(* Logix 5000 project; controller cal1632 1756-L62 rev 16.20; software revision 16.05; part 56 of 57 *)
(* tags used below, declared in another part *)
   FAULT : BOOL;
   HMI : BOOL;
   p01r09_pb_global_reset : BOOL;
   p30_di_pin_1 : BOOL;
   p30_di_pin_2 : BOOL;
   p30_di_pin_3 : BOOL;
   p30_di_pin_4 : BOOL;
   p30_di_pin_5 : BOOL;
   p30_di_pin_6 : BOOL;
   p30_di_pin_7 : BOOL;
   p30_di_pin_8 : BOOL;
   p30_dint_to_hmi : DINT[16];
   p30_do_retract_motion : BOOL;
   p30_do_rotation_fwd : BOOL;
   p30_do_rotation_rev : BOOL;
   p30_real_to_hmi : REAL[112];
   p30r04 : routine;
   p30r04_timer_fault : TIMER[4];
   p30r04_timer_warning : TIMER[4];
   p30r05 : routine;
   p30r05_timer_fault : TIMER[4];
   p30r05_timer_warning : TIMER[4];
   p30r06 : routine;
   p30r06_timer_fault : TIMER[4];
   p30r06_timer_warning : TIMER[4];
   p30r07 : routine;
   p30r07_timer_fault : TIMER[4];
   p30r07_timer_warning : TIMER[4];
   p30r10 : routine;
(* P30_Retraction_System, continued *)

ROUTINE R04_Output   (* ladder *)
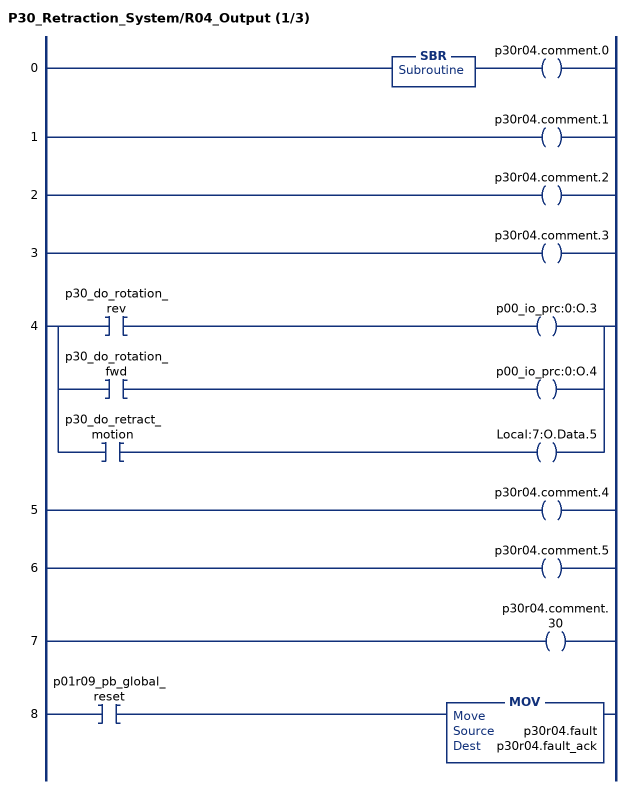
   0: SBR()OTE(p30r04.comment.0);
   1: OTE(p30r04.comment.1);
   2: OTE(p30r04.comment.2);
   3: OTE(p30r04.comment.3);
   4: [XIC(p30_do_rotation_rev) OTE(p00_io_prc:0:O.3) ,XIC(p30_do_rotation_fwd) OTE(p00_io_prc:0:O.4) ,XIC(p30_do_retract_motion) OTE(Local:7:O.Data.5) ];
   5: OTE(p30r04.comment.4);
   6: OTE(p30r04.comment.5);
   7: OTE(p30r04.comment.30);
   8: XIC(p01r09_pb_global_reset)MOV(p30r04.fault,p30r04.fault_ack);
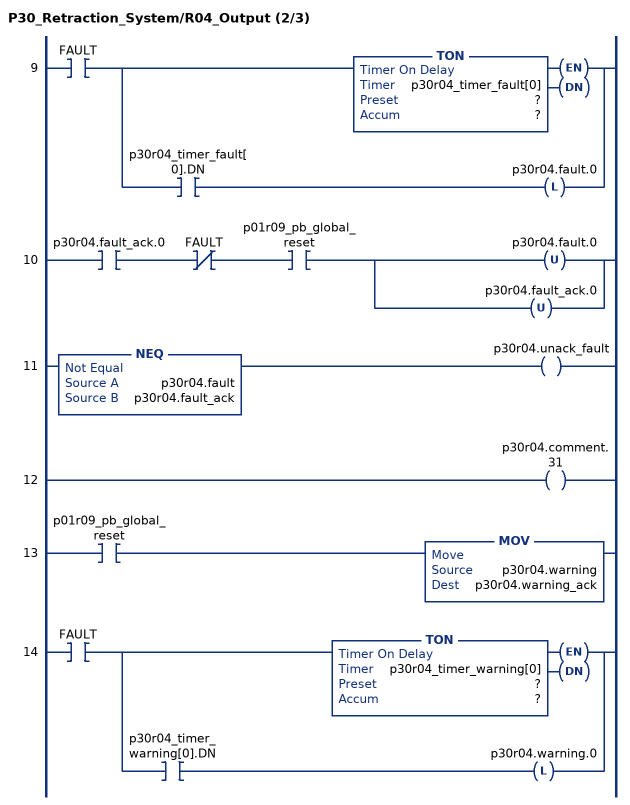
   9: XIC(FAULT)[TON(p30r04_timer_fault[0],?,?) ,XIC(p30r04_timer_fault[0].DN) OTL(p30r04.fault.0) ];
   10: XIC(p30r04.fault_ack.0)XIO(FAULT)XIC(p01r09_pb_global_reset)[OTU(p30r04.fault.0) ,OTU(p30r04.fault_ack.0) ];
   11: NEQ(p30r04.fault,p30r04.fault_ack)OTE(p30r04.unack_fault);
   12: OTE(p30r04.comment.31);
   13: XIC(p01r09_pb_global_reset)MOV(p30r04.warning,p30r04.warning_ack);
   14: XIC(FAULT)[TON(p30r04_timer_warning[0],?,?) ,XIC(p30r04_timer_warning[0].DN) OTL(p30r04.warning.0) ];
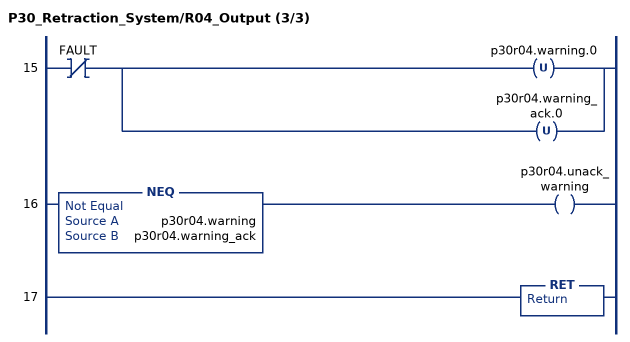
   15: XIO(FAULT)[OTU(p30r04.warning.0) ,OTU(p30r04.warning_ack.0) ];
   16: NEQ(p30r04.warning,p30r04.warning_ack)OTE(p30r04.unack_warning);
   17: RET();
END_ROUTINE

ROUTINE R05_Dint_to_HMI   (* ladder *)
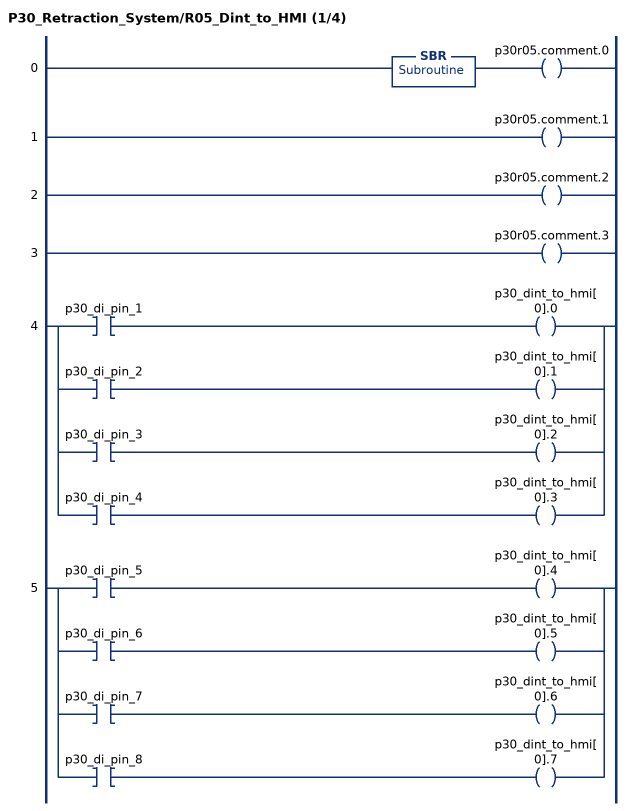
   0: SBR()OTE(p30r05.comment.0);
   1: OTE(p30r05.comment.1);
   2: OTE(p30r05.comment.2);
   3: OTE(p30r05.comment.3);
   4: [XIC(p30_di_pin_1) OTE(p30_dint_to_hmi[0].0) ,XIC(p30_di_pin_2) OTE(p30_dint_to_hmi[0].1) ,XIC(p30_di_pin_3) OTE(p30_dint_to_hmi[0].2) ,XIC(p30_di_pin_4) OTE(p30_dint_to_hmi[0].3) ];
   5: [XIC(p30_di_pin_5) OTE(p30_dint_to_hmi[0].4) ,XIC(p30_di_pin_6) OTE(p30_dint_to_hmi[0].5) ,XIC(p30_di_pin_7) OTE(p30_dint_to_hmi[0].6) ,XIC(p30_di_pin_8) OTE(p30_dint_to_hmi[0].7) ];
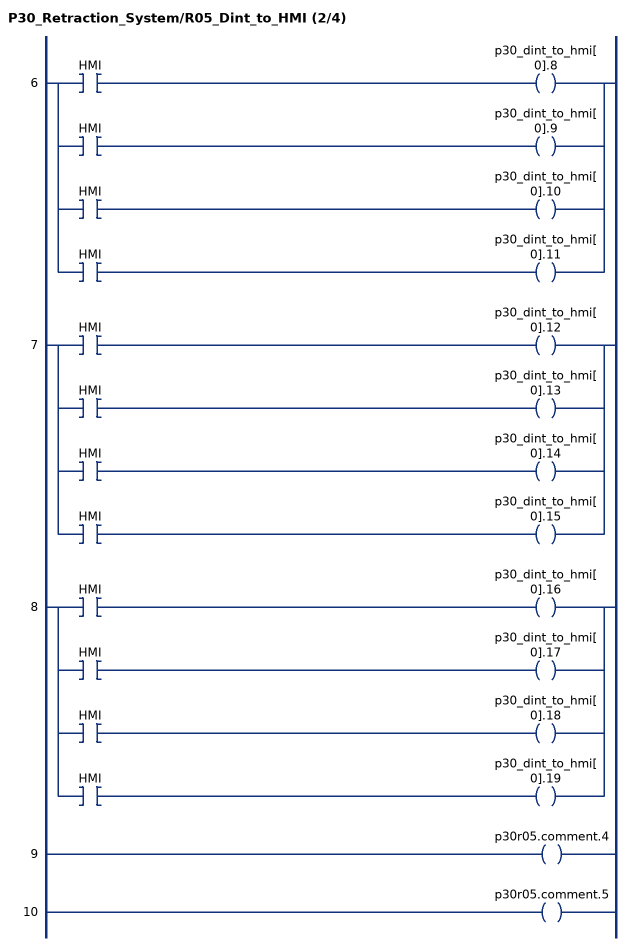
   6: [XIC(HMI) OTE(p30_dint_to_hmi[0].8) ,XIC(HMI) OTE(p30_dint_to_hmi[0].9) ,XIC(HMI) OTE(p30_dint_to_hmi[0].10) ,XIC(HMI) OTE(p30_dint_to_hmi[0].11) ];
   7: [XIC(HMI) OTE(p30_dint_to_hmi[0].12) ,XIC(HMI) OTE(p30_dint_to_hmi[0].13) ,XIC(HMI) OTE(p30_dint_to_hmi[0].14) ,XIC(HMI) OTE(p30_dint_to_hmi[0].15) ];
   8: [XIC(HMI) OTE(p30_dint_to_hmi[0].16) ,XIC(HMI) OTE(p30_dint_to_hmi[0].17) ,XIC(HMI) OTE(p30_dint_to_hmi[0].18) ,XIC(HMI) OTE(p30_dint_to_hmi[0].19) ];
   9: OTE(p30r05.comment.4);
   10: OTE(p30r05.comment.5);
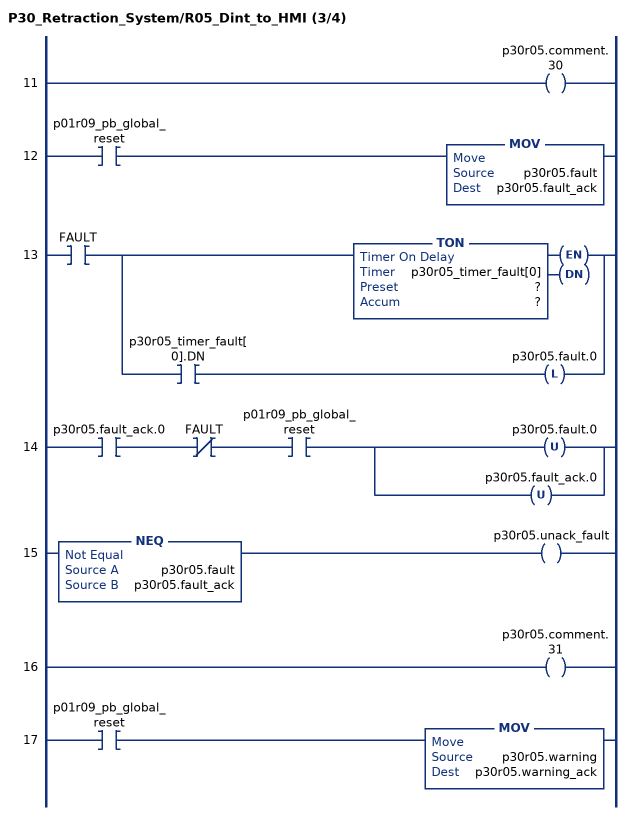
   11: OTE(p30r05.comment.30);
   12: XIC(p01r09_pb_global_reset)MOV(p30r05.fault,p30r05.fault_ack);
   13: XIC(FAULT)[TON(p30r05_timer_fault[0],?,?) ,XIC(p30r05_timer_fault[0].DN) OTL(p30r05.fault.0) ];
   14: XIC(p30r05.fault_ack.0)XIO(FAULT)XIC(p01r09_pb_global_reset)[OTU(p30r05.fault.0) ,OTU(p30r05.fault_ack.0) ];
   15: NEQ(p30r05.fault,p30r05.fault_ack)OTE(p30r05.unack_fault);
   16: OTE(p30r05.comment.31);
   17: XIC(p01r09_pb_global_reset)MOV(p30r05.warning,p30r05.warning_ack);
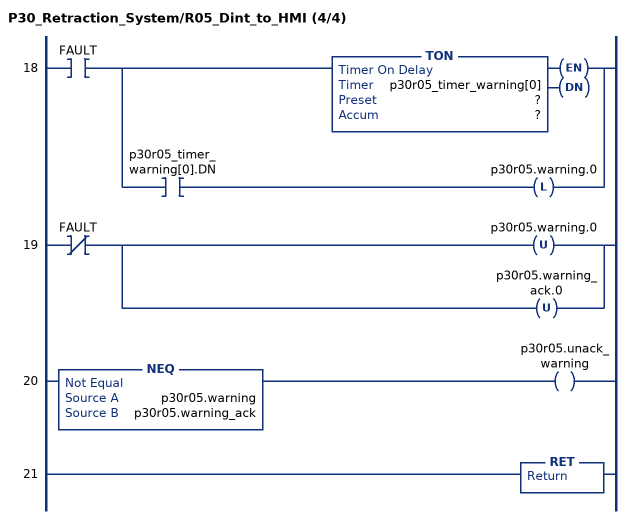
   18: XIC(FAULT)[TON(p30r05_timer_warning[0],?,?) ,XIC(p30r05_timer_warning[0].DN) OTL(p30r05.warning.0) ];
   19: XIO(FAULT)[OTU(p30r05.warning.0) ,OTU(p30r05.warning_ack.0) ];
   20: NEQ(p30r05.warning,p30r05.warning_ack)OTE(p30r05.unack_warning);
   21: RET();
END_ROUTINE

ROUTINE R06_Real_to_HMI   (* ladder *)
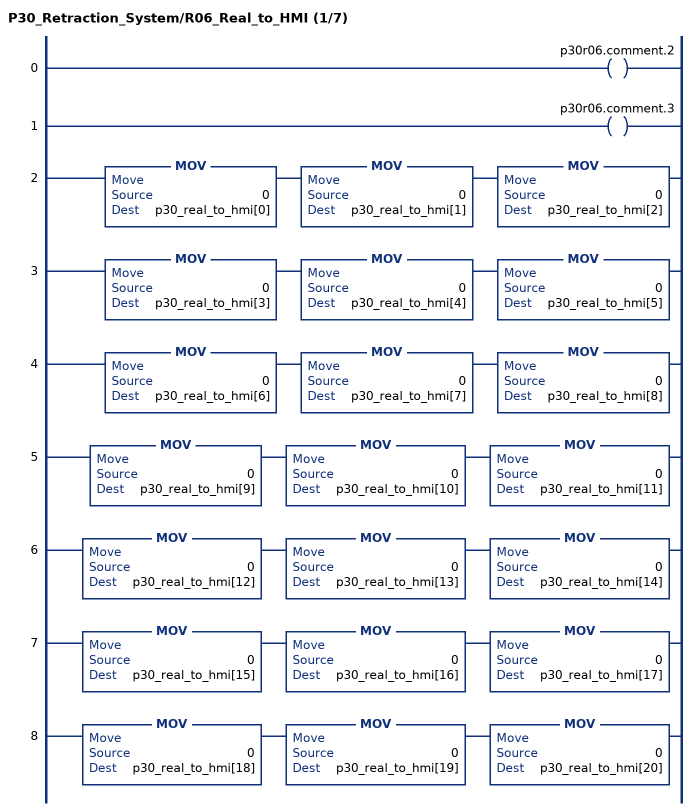
   0: OTE(p30r06.comment.2);
   1: OTE(p30r06.comment.3);
   2: MOV(0,p30_real_to_hmi[0])MOV(0,p30_real_to_hmi[1])MOV(0,p30_real_to_hmi[2]);
   3: MOV(0,p30_real_to_hmi[3])MOV(0,p30_real_to_hmi[4])MOV(0,p30_real_to_hmi[5]);
   4: MOV(0,p30_real_to_hmi[6])MOV(0,p30_real_to_hmi[7])MOV(0,p30_real_to_hmi[8]);
   5: MOV(0,p30_real_to_hmi[9])MOV(0,p30_real_to_hmi[10])MOV(0,p30_real_to_hmi[11]);
   6: MOV(0,p30_real_to_hmi[12])MOV(0,p30_real_to_hmi[13])MOV(0,p30_real_to_hmi[14]);
   7: MOV(0,p30_real_to_hmi[15])MOV(0,p30_real_to_hmi[16])MOV(0,p30_real_to_hmi[17]);
   8: MOV(0,p30_real_to_hmi[18])MOV(0,p30_real_to_hmi[19])MOV(0,p30_real_to_hmi[20]);
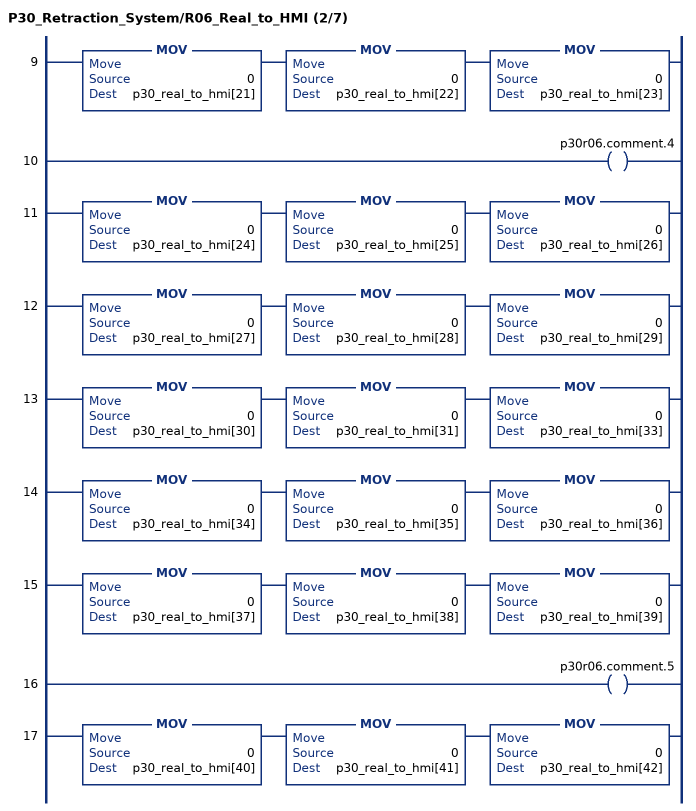
   9: MOV(0,p30_real_to_hmi[21])MOV(0,p30_real_to_hmi[22])MOV(0,p30_real_to_hmi[23]);
   10: OTE(p30r06.comment.4);
   11: MOV(0,p30_real_to_hmi[24])MOV(0,p30_real_to_hmi[25])MOV(0,p30_real_to_hmi[26]);
   12: MOV(0,p30_real_to_hmi[27])MOV(0,p30_real_to_hmi[28])MOV(0,p30_real_to_hmi[29]);
   13: MOV(0,p30_real_to_hmi[30])MOV(0,p30_real_to_hmi[31])MOV(0,p30_real_to_hmi[33]);
   14: MOV(0,p30_real_to_hmi[34])MOV(0,p30_real_to_hmi[35])MOV(0,p30_real_to_hmi[36]);
   15: MOV(0,p30_real_to_hmi[37])MOV(0,p30_real_to_hmi[38])MOV(0,p30_real_to_hmi[39]);
   16: OTE(p30r06.comment.5);
   17: MOV(0,p30_real_to_hmi[40])MOV(0,p30_real_to_hmi[41])MOV(0,p30_real_to_hmi[42]);
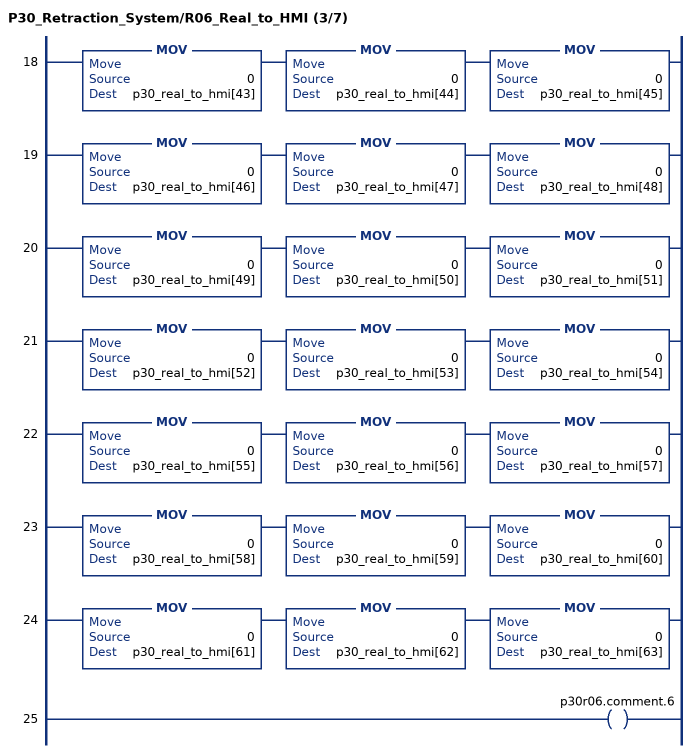
   18: MOV(0,p30_real_to_hmi[43])MOV(0,p30_real_to_hmi[44])MOV(0,p30_real_to_hmi[45]);
   19: MOV(0,p30_real_to_hmi[46])MOV(0,p30_real_to_hmi[47])MOV(0,p30_real_to_hmi[48]);
   20: MOV(0,p30_real_to_hmi[49])MOV(0,p30_real_to_hmi[50])MOV(0,p30_real_to_hmi[51]);
   21: MOV(0,p30_real_to_hmi[52])MOV(0,p30_real_to_hmi[53])MOV(0,p30_real_to_hmi[54]);
   22: MOV(0,p30_real_to_hmi[55])MOV(0,p30_real_to_hmi[56])MOV(0,p30_real_to_hmi[57]);
   23: MOV(0,p30_real_to_hmi[58])MOV(0,p30_real_to_hmi[59])MOV(0,p30_real_to_hmi[60]);
   24: MOV(0,p30_real_to_hmi[61])MOV(0,p30_real_to_hmi[62])MOV(0,p30_real_to_hmi[63]);
   25: OTE(p30r06.comment.6);
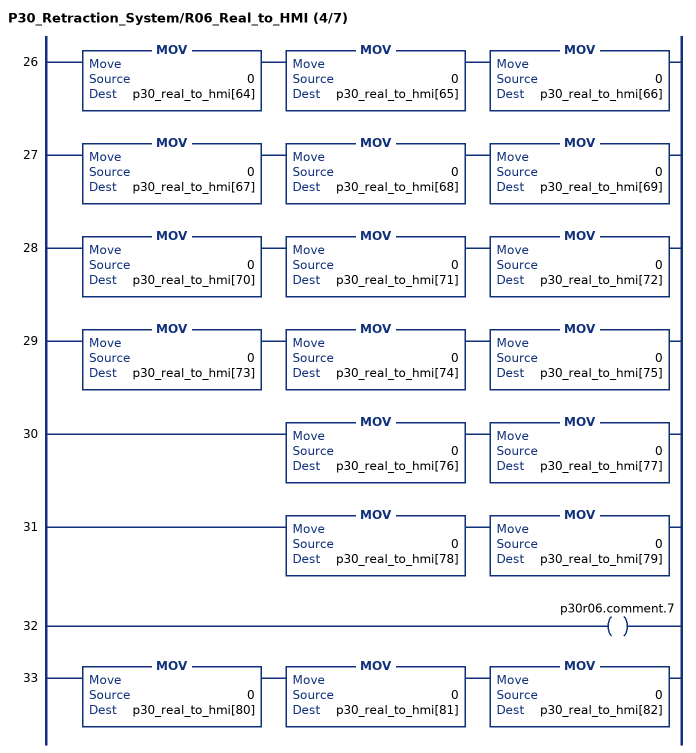
   26: MOV(0,p30_real_to_hmi[64])MOV(0,p30_real_to_hmi[65])MOV(0,p30_real_to_hmi[66]);
   27: MOV(0,p30_real_to_hmi[67])MOV(0,p30_real_to_hmi[68])MOV(0,p30_real_to_hmi[69]);
   28: MOV(0,p30_real_to_hmi[70])MOV(0,p30_real_to_hmi[71])MOV(0,p30_real_to_hmi[72]);
   29: MOV(0,p30_real_to_hmi[73])MOV(0,p30_real_to_hmi[74])MOV(0,p30_real_to_hmi[75]);
   30: MOV(0,p30_real_to_hmi[76])MOV(0,p30_real_to_hmi[77]);
   31: MOV(0,p30_real_to_hmi[78])MOV(0,p30_real_to_hmi[79]);
   32: OTE(p30r06.comment.7);
   33: MOV(0,p30_real_to_hmi[80])MOV(0,p30_real_to_hmi[81])MOV(0,p30_real_to_hmi[82]);
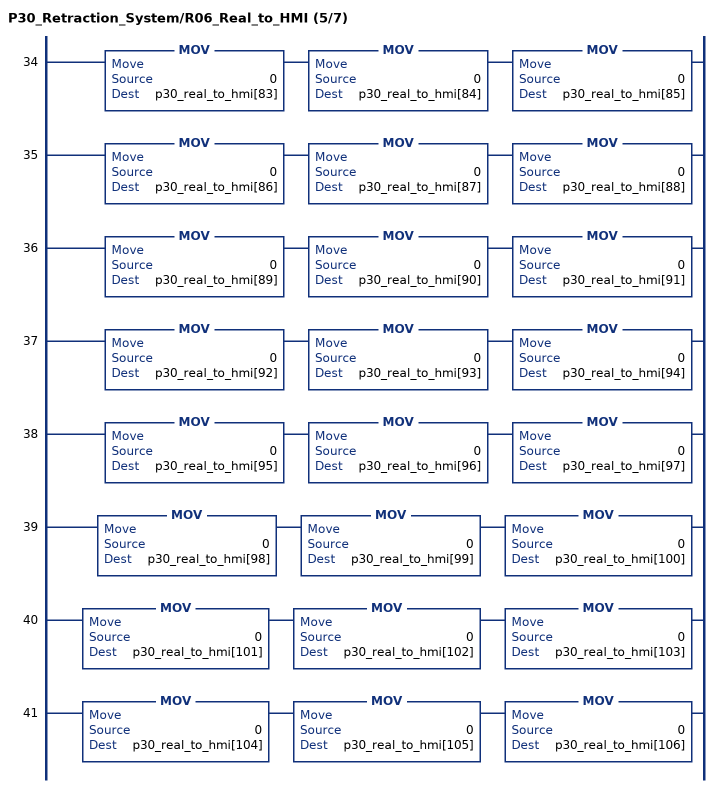
   34: MOV(0,p30_real_to_hmi[83])MOV(0,p30_real_to_hmi[84])MOV(0,p30_real_to_hmi[85]);
   35: MOV(0,p30_real_to_hmi[86])MOV(0,p30_real_to_hmi[87])MOV(0,p30_real_to_hmi[88]);
   36: MOV(0,p30_real_to_hmi[89])MOV(0,p30_real_to_hmi[90])MOV(0,p30_real_to_hmi[91]);
   37: MOV(0,p30_real_to_hmi[92])MOV(0,p30_real_to_hmi[93])MOV(0,p30_real_to_hmi[94]);
   38: MOV(0,p30_real_to_hmi[95])MOV(0,p30_real_to_hmi[96])MOV(0,p30_real_to_hmi[97]);
   39: MOV(0,p30_real_to_hmi[98])MOV(0,p30_real_to_hmi[99])MOV(0,p30_real_to_hmi[100]);
   40: MOV(0,p30_real_to_hmi[101])MOV(0,p30_real_to_hmi[102])MOV(0,p30_real_to_hmi[103]);
   41: MOV(0,p30_real_to_hmi[104])MOV(0,p30_real_to_hmi[105])MOV(0,p30_real_to_hmi[106]);
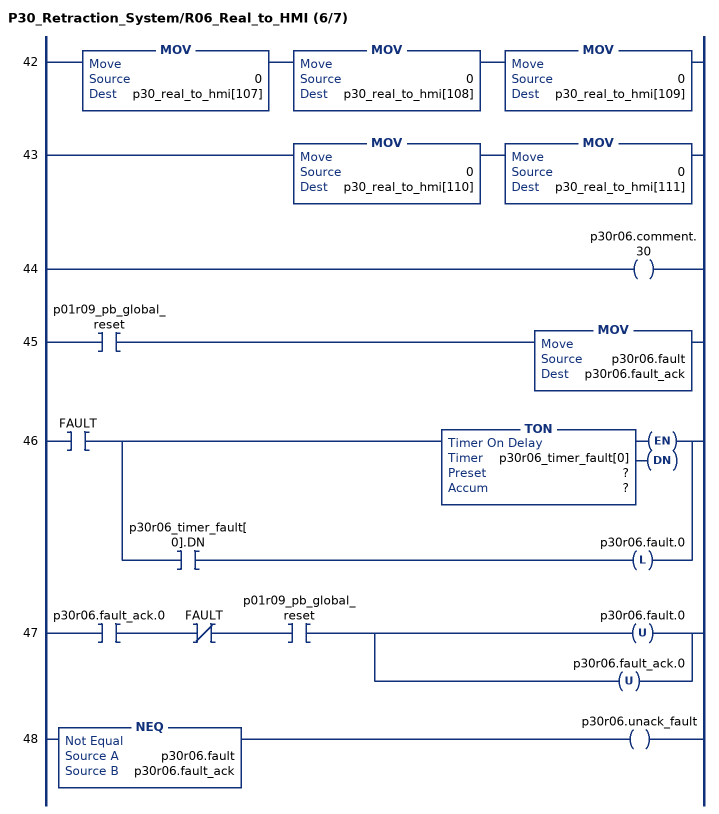
   42: MOV(0,p30_real_to_hmi[107])MOV(0,p30_real_to_hmi[108])MOV(0,p30_real_to_hmi[109]);
   43: MOV(0,p30_real_to_hmi[110])MOV(0,p30_real_to_hmi[111]);
   44: OTE(p30r06.comment.30);
   45: XIC(p01r09_pb_global_reset)MOV(p30r06.fault,p30r06.fault_ack);
   46: XIC(FAULT)[TON(p30r06_timer_fault[0],?,?) ,XIC(p30r06_timer_fault[0].DN) OTL(p30r06.fault.0) ];
   47: XIC(p30r06.fault_ack.0)XIO(FAULT)XIC(p01r09_pb_global_reset)[OTU(p30r06.fault.0) ,OTU(p30r06.fault_ack.0) ];
   48: NEQ(p30r06.fault,p30r06.fault_ack)OTE(p30r06.unack_fault);
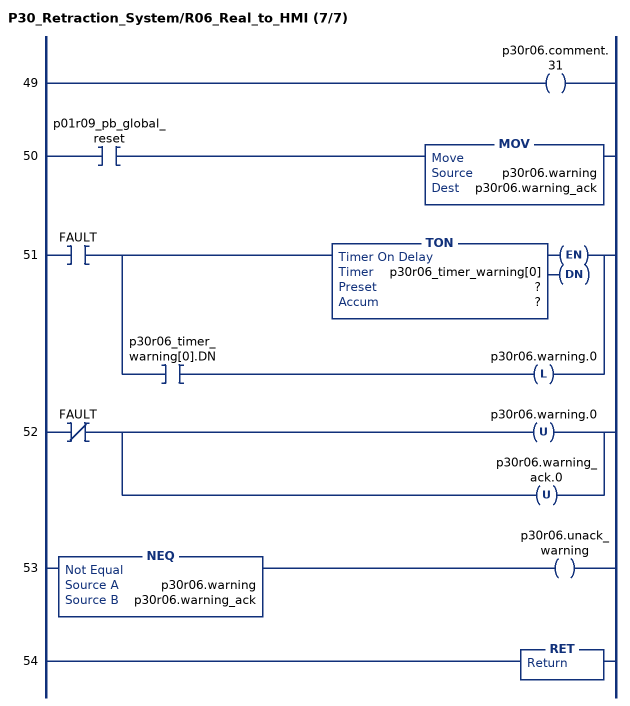
   49: OTE(p30r06.comment.31);
   50: XIC(p01r09_pb_global_reset)MOV(p30r06.warning,p30r06.warning_ack);
   51: XIC(FAULT)[TON(p30r06_timer_warning[0],?,?) ,XIC(p30r06_timer_warning[0].DN) OTL(p30r06.warning.0) ];
   52: XIO(FAULT)[OTU(p30r06.warning.0) ,OTU(p30r06.warning_ack.0) ];
   53: NEQ(p30r06.warning,p30r06.warning_ack)OTE(p30r06.unack_warning);
   54: RET();
END_ROUTINE

ROUTINE R07_Alarms   (* ladder *)
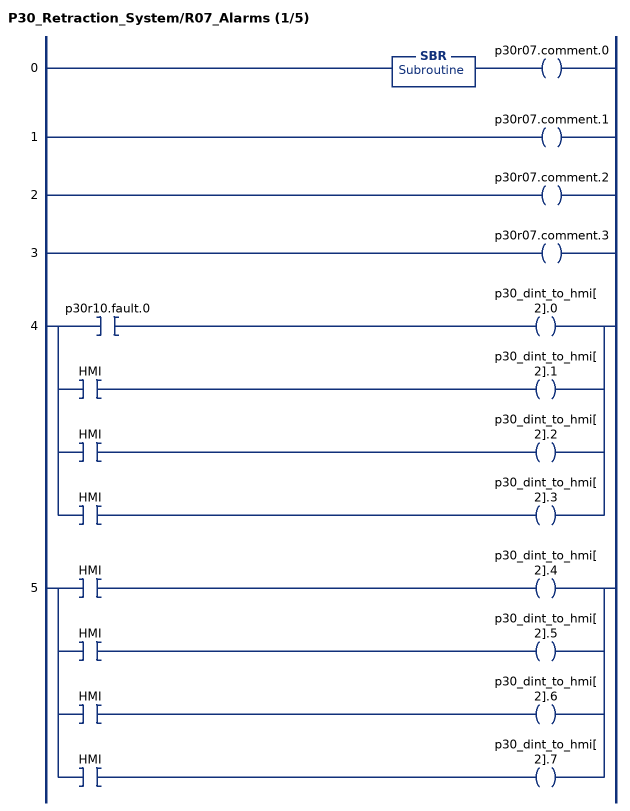
   0: SBR()OTE(p30r07.comment.0);
   1: OTE(p30r07.comment.1);
   2: OTE(p30r07.comment.2);
   3: OTE(p30r07.comment.3);
   4: [XIC(p30r10.fault.0) OTE(p30_dint_to_hmi[2].0) ,XIC(HMI) OTE(p30_dint_to_hmi[2].1) ,XIC(HMI) OTE(p30_dint_to_hmi[2].2) ,XIC(HMI) OTE(p30_dint_to_hmi[2].3) ];
   5: [XIC(HMI) OTE(p30_dint_to_hmi[2].4) ,XIC(HMI) OTE(p30_dint_to_hmi[2].5) ,XIC(HMI) OTE(p30_dint_to_hmi[2].6) ,XIC(HMI) OTE(p30_dint_to_hmi[2].7) ];
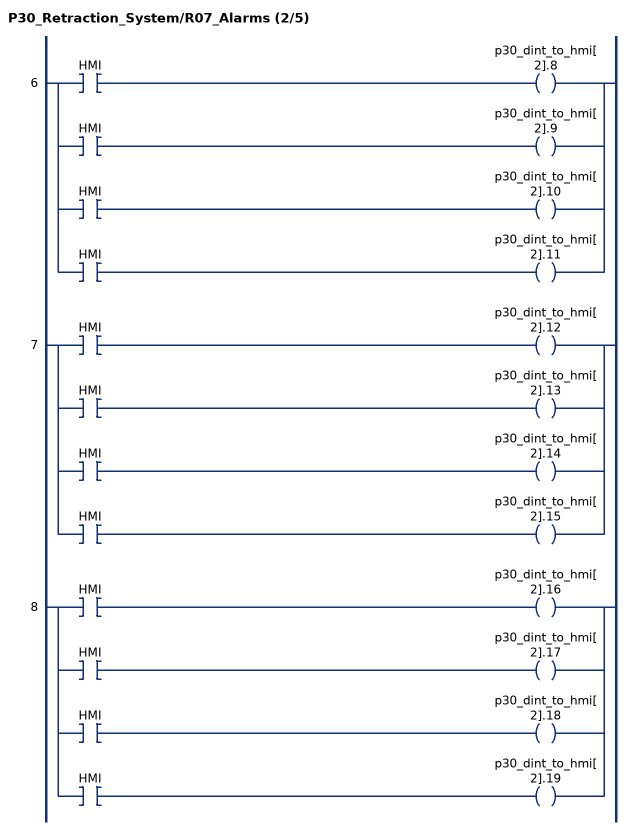
   6: [XIC(HMI) OTE(p30_dint_to_hmi[2].8) ,XIC(HMI) OTE(p30_dint_to_hmi[2].9) ,XIC(HMI) OTE(p30_dint_to_hmi[2].10) ,XIC(HMI) OTE(p30_dint_to_hmi[2].11) ];
   7: [XIC(HMI) OTE(p30_dint_to_hmi[2].12) ,XIC(HMI) OTE(p30_dint_to_hmi[2].13) ,XIC(HMI) OTE(p30_dint_to_hmi[2].14) ,XIC(HMI) OTE(p30_dint_to_hmi[2].15) ];
   8: [XIC(HMI) OTE(p30_dint_to_hmi[2].16) ,XIC(HMI) OTE(p30_dint_to_hmi[2].17) ,XIC(HMI) OTE(p30_dint_to_hmi[2].18) ,XIC(HMI) OTE(p30_dint_to_hmi[2].19) ];
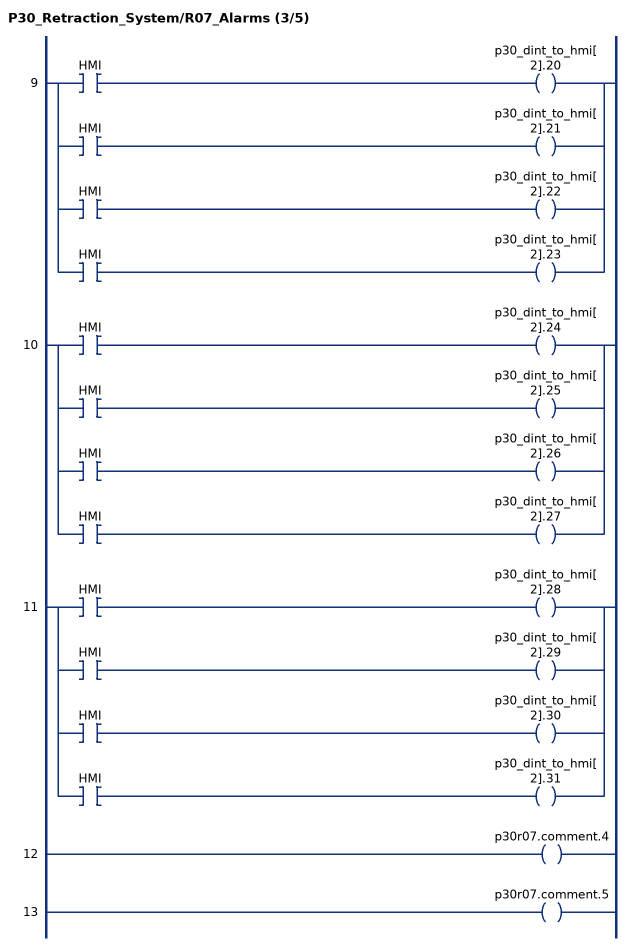
   9: [XIC(HMI) OTE(p30_dint_to_hmi[2].20) ,XIC(HMI) OTE(p30_dint_to_hmi[2].21) ,XIC(HMI) OTE(p30_dint_to_hmi[2].22) ,XIC(HMI) OTE(p30_dint_to_hmi[2].23) ];
   10: [XIC(HMI) OTE(p30_dint_to_hmi[2].24) ,XIC(HMI) OTE(p30_dint_to_hmi[2].25) ,XIC(HMI) OTE(p30_dint_to_hmi[2].26) ,XIC(HMI) OTE(p30_dint_to_hmi[2].27) ];
   11: [XIC(HMI) OTE(p30_dint_to_hmi[2].28) ,XIC(HMI) OTE(p30_dint_to_hmi[2].29) ,XIC(HMI) OTE(p30_dint_to_hmi[2].30) ,XIC(HMI) OTE(p30_dint_to_hmi[2].31) ];
   12: OTE(p30r07.comment.4);
   13: OTE(p30r07.comment.5);
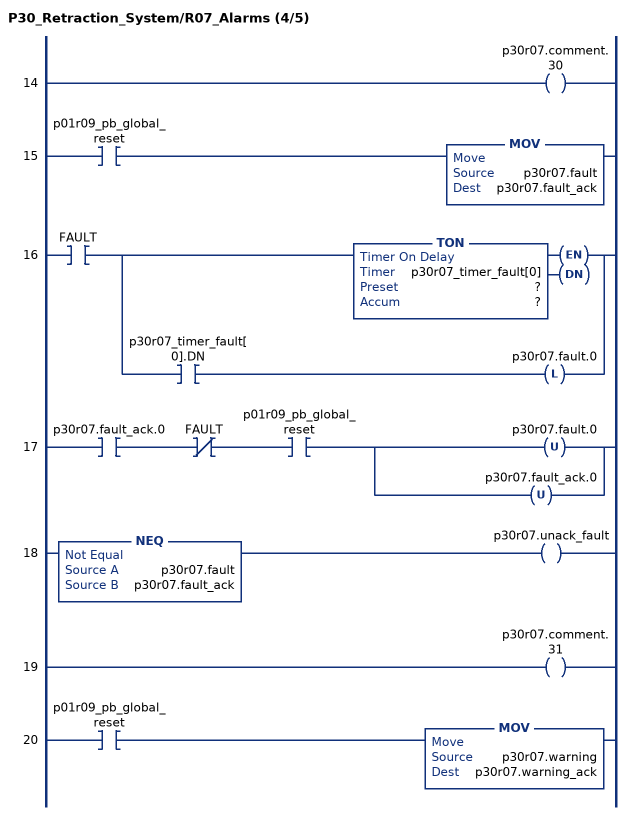
   14: OTE(p30r07.comment.30);
   15: XIC(p01r09_pb_global_reset)MOV(p30r07.fault,p30r07.fault_ack);
   16: XIC(FAULT)[TON(p30r07_timer_fault[0],?,?) ,XIC(p30r07_timer_fault[0].DN) OTL(p30r07.fault.0) ];
   17: XIC(p30r07.fault_ack.0)XIO(FAULT)XIC(p01r09_pb_global_reset)[OTU(p30r07.fault.0) ,OTU(p30r07.fault_ack.0) ];
   18: NEQ(p30r07.fault,p30r07.fault_ack)OTE(p30r07.unack_fault);
   19: OTE(p30r07.comment.31);
   20: XIC(p01r09_pb_global_reset)MOV(p30r07.warning,p30r07.warning_ack);
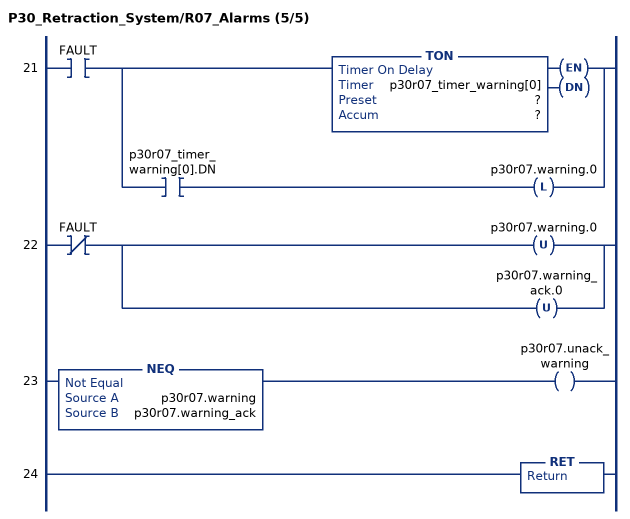
   21: XIC(FAULT)[TON(p30r07_timer_warning[0],?,?) ,XIC(p30r07_timer_warning[0].DN) OTL(p30r07.warning.0) ];
   22: XIO(FAULT)[OTU(p30r07.warning.0) ,OTU(p30r07.warning_ack.0) ];
   23: NEQ(p30r07.warning,p30r07.warning_ack)OTE(p30r07.unack_warning);
   24: RET();
END_ROUTINE
